Yaskawa INFORM job: MALBEN3.JBI

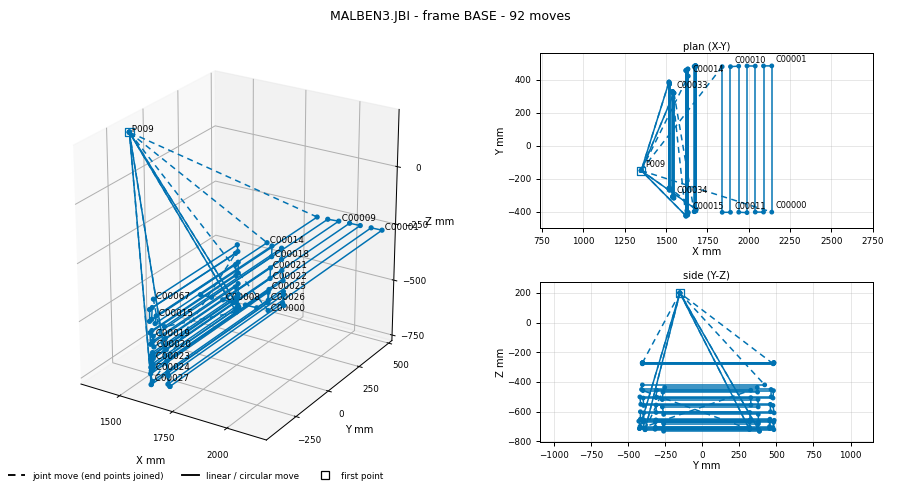
[picture p0: tool path of MALBEN3.JBI in frame BASE, 92 of 92 moves have a stored position in this frame; points joined in program order, loops and branches not executed]
/JOB
//NAME MALBEN3
//POS
///NPOS 86,0,86,1,0,1
///TOOL 0
///POSTYPE BASE
///RECTAN
///RCONF 1,0,0,0,0,0,0,0,0,0,0,0,0,0,0,0,0,0,0,0,0,0,0,0
C00000=2140.098,-401.360,-268.977,175.0000,5.0000,5.0000
C00001=2140.098,483.583,-268.977,175.0000,5.0000,5.0000
C00002=2090.098,483.455,-270.030,175.0000,5.0000,5.0000
C00003=2090.098,-401.273,-270.030,175.0000,5.0000,5.0000
C00004=2040.098,-401.141,-271.239,175.0000,5.0000,5.0000
C00005=2040.098,482.568,-271.239,175.0000,5.0000,5.0000
C00006=1990.098,483.262,-272.654,175.0000,5.0000,5.0000
C00007=1990.098,-404.579,-272.654,175.0000,5.0000,5.0000
C00008=1940.098,-401.886,-274.425,175.0000,5.0000,5.0000
C00009=1940.098,482.155,-274.425,175.0000,5.0000,5.0000
C00010=1890.098,478.954,-276.250,175.0000,5.0000,5.0000
C00011=1890.098,-402.510,-276.250,175.0000,5.0000,5.0000
C00012=1839.960,-402.553,-277.742,175.0000,5.0000,5.0000
C00013=1839.960,478.937,-277.742,175.0000,5.0000,5.0000
C00014=1634.901,421.672,-419.637,175.0000,-89.9999,5.0000
C00015=1634.901,-402.743,-419.637,175.0000,-89.9999,5.0000
C00016=1633.143,-408.452,-450.789,175.0000,-89.9999,5.0000
C00017=1633.143,464.348,-450.789,175.0000,-89.9999,5.0000
C00018=1631.374,465.131,-500.789,175.0000,-89.9999,5.0000
C00019=1631.374,-419.852,-500.789,175.0000,-89.9999,5.0000
C00020=1629.352,-413.747,-550.789,175.0000,-89.9999,5.0000
C00021=1629.352,459.427,-550.789,175.0000,-89.9999,5.0000
C00022=1626.911,460.715,-600.789,175.0000,-89.9999,5.0000
C00023=1626.911,-416.191,-600.789,175.0000,-89.9999,5.0000
C00024=1624.499,-416.100,-650.789,175.0000,-89.9999,5.0000
C00025=1624.499,456.978,-650.789,175.0000,-89.9999,5.0000
C00026=1622.503,454.505,-700.789,175.0000,-89.9999,5.0000
C00027=1622.503,-418.968,-700.789,175.0000,-89.9999,5.0000
C00028=1620.879,-427.008,-664.187,180.0000,-60.0000,0.0000
C00029=1620.879,455.687,-664.187,180.0000,-60.0000,0.0000
C00030=1619.373,455.631,-714.187,180.0000,-60.0000,0.0000
C00031=1619.373,-422.309,-714.187,180.0000,-60.0000,0.0000
C00032=1619.373,-422.309,-714.187,180.0000,-60.0000,0.0000
C00033=1538.648,327.998,-455.742,175.0000,-89.9999,5.0000
C00034=1538.648,-307.231,-455.742,175.0000,-89.9999,5.0000
C00035=1539.732,-310.347,-505.742,175.0000,-89.9999,5.0000
C00036=1539.732,327.893,-505.742,175.0000,-89.9999,5.0000
C00037=1540.970,328.259,-555.742,175.0000,-89.9999,5.0000
C00038=1540.970,-310.206,-555.742,175.0000,-89.9999,5.0000
C00039=1542.330,-310.096,-605.742,175.0000,-89.9999,5.0000
C00040=1542.330,320.907,-605.742,175.0000,-89.9999,5.0000
C00041=1543.566,323.502,-655.742,175.0000,-89.9999,5.0000
C00042=1543.566,-311.381,-655.742,175.0000,-89.9999,5.0000
C00043=1545.116,-315.143,-705.742,175.0000,-89.9999,5.0000
C00044=1545.116,319.629,-705.742,175.0000,-89.9999,5.0000
C00045=1546.765,320.274,-669.140,180.0000,-60.0000,0.0000
C00046=1546.765,-315.233,-669.140,180.0000,-60.0000,0.0000
C00047=1548.154,-316.980,-719.140,180.0000,-60.0000,0.0000
C00048=1548.154,319.087,-719.140,180.0000,-60.0000,0.0000
C00049=1548.154,319.087,-719.140,180.0000,-60.0000,0.0000
C00050=1670.216,-398.864,-458.454,175.0000,-89.9999,5.0000
C00051=1670.216,480.762,-458.454,175.0000,-89.9999,5.0000
C00052=1672.445,477.562,-508.454,175.0000,-89.9999,5.0000
C00053=1672.445,-397.223,-508.454,175.0000,-89.9999,5.0000
C00054=1674.551,-394.686,-558.454,175.0000,-89.9999,5.0000
C00055=1674.551,477.382,-558.454,175.0000,-89.9999,5.0000
C00056=1676.296,485.126,-608.454,175.0000,-89.9999,5.0000
C00057=1676.296,-393.486,-608.454,175.0000,-89.9999,5.0000
C00058=1677.899,-392.919,-658.454,175.0000,-89.9999,5.0000
C00059=1677.899,485.748,-658.454,175.0000,-89.9999,5.0000
C00060=1679.509,477.056,-708.454,175.0000,-89.9999,5.0000
C00061=1679.509,-394.482,-708.454,175.0000,-89.9999,5.0000
C00062=1680.701,-393.512,-671.851,180.0000,-60.0000,0.0000
C00063=1680.701,481.956,-671.851,180.0000,-60.0000,0.0000
C00064=1682.129,483.373,-721.851,180.0000,-60.0000,0.0000
C00065=1682.129,-384.577,-721.851,180.0000,-60.0000,0.0000
C00066=1682.129,-384.577,-721.851,180.0000,-60.0000,0.0000
C00067=1520.388,-252.750,-437.009,175.0000,-89.9999,5.0000
C00068=1520.388,371.413,-437.009,175.0000,-89.9999,5.0000
C00069=1521.796,373.507,-468.529,175.0000,-89.9999,5.0000
C00070=1521.796,-264.209,-468.529,175.0000,-89.9999,5.0000
C00071=1521.398,-268.886,-518.529,175.0000,-89.9999,5.0000
C00072=1521.398,376.643,-518.529,175.0000,-89.9999,5.0000
C00073=1521.017,377.744,-568.529,175.0000,-89.9999,5.0000
C00074=1521.017,-268.182,-568.529,175.0000,-89.9999,5.0000
C00075=1519.841,-259.271,-618.529,175.0000,-89.9999,5.0000
C00076=1519.841,378.499,-618.529,175.0000,-89.9999,5.0000
C00077=1519.405,379.693,-668.529,175.0000,-89.9999,5.0000
C00078=1519.405,-263.625,-668.529,175.0000,-89.9999,5.0000
C00079=1519.161,-262.870,-718.529,175.0000,-89.9999,5.0000
C00080=1519.161,378.578,-718.529,175.0000,-89.9999,5.0000
C00081=1518.693,379.125,-681.927,180.0000,-60.0000,0.0000
C00082=1518.693,-258.984,-681.927,180.0000,-60.0000,0.0000
C00083=1518.160,-259.608,-731.927,180.0000,-60.0000,0.0000
C00084=1518.160,386.235,-731.927,180.0000,-60.0000,0.0000
C00085=1518.160,386.235,-731.927,180.0000,-60.0000,0.0000
///POSTYPE PULSE
///PULSE
EC00000=0
EC00001=0
EC00002=0
EC00003=0
EC00004=0
EC00005=0
EC00006=0
EC00007=0
EC00008=0
EC00009=0
EC00010=0
EC00011=0
EC00012=0
EC00013=0
EC00014=0
EC00015=0
EC00016=0
EC00017=0
EC00018=0
EC00019=0
EC00020=0
EC00021=0
EC00022=0
EC00023=0
EC00024=0
EC00025=0
EC00026=0
EC00027=0
EC00028=0
EC00029=0
EC00030=0
EC00031=0
EC00032=92160
EC00033=92160
EC00034=92160
EC00035=92160
EC00036=92160
EC00037=92160
EC00038=92160
EC00039=92160
EC00040=92160
EC00041=92160
EC00042=92160
EC00043=92160
EC00044=92160
EC00045=92160
EC00046=92160
EC00047=92160
EC00048=92160
EC00049=184320
EC00050=184320
EC00051=184320
EC00052=184320
EC00053=184320
EC00054=184320
EC00055=184320
EC00056=184320
EC00057=184320
EC00058=184320
EC00059=184320
EC00060=184320
EC00061=184320
EC00062=184320
EC00063=184320
EC00064=184320
EC00065=184320
EC00066=276480
EC00067=276480
EC00068=276480
EC00069=276480
EC00070=276480
EC00071=276480
EC00072=276480
EC00073=276480
EC00074=276480
EC00075=276480
EC00076=276480
EC00077=276480
EC00078=276480
EC00079=276480
EC00080=276480
EC00081=276480
EC00082=276480
EC00083=276480
EC00084=276480
EC00085=368640
///POSTYPE BASE
///RECTAN
P00009=1350.000,-150.000,200.000,-180.0000,-45.0000,0.0000
///POSTYPE PULSE
///PULSE
EX00000=0
//INST
///DATE 2023/03/14 16:30
///ATTR SC,RW,RJ
////FRAME BASE
///GROUP1 RB1,ST1
NOP
MOVJ P009 EX000 VJ=15.00
MOVJ C00000 EC00000 VJ=15.00
CALL JOB:SPYON
MOVL C00001 EC00001 V=150.0
MOVL C00002 EC00002 V=150.0
MOVL C00003 EC00003 V=150.0
MOVL C00004 EC00004 V=150.0
MOVL C00005 EC00005 V=150.0
MOVL C00006 EC00006 V=150.0
MOVL C00007 EC00007 V=150.0
MOVL C00008 EC00008 V=150.0
MOVL C00009 EC00009 V=150.0
MOVL C00010 EC00010 V=150.0
MOVL C00011 EC00011 V=150.0
MOVL C00012 EC00012 V=150.0
MOVL C00013 EC00013 V=150.0
CALL JOB:SPYOF
MOVJ P009 VJ=15.00
MOVJ C00014 EC00014 VJ=15.00
CALL JOB:SPYON
MOVL C00015 EC00015 V=150.0
MOVL C00016 EC00016 V=150.0
MOVL C00017 EC00017 V=150.0
MOVL C00018 EC00018 V=150.0
MOVL C00019 EC00019 V=150.0
MOVL C00020 EC00020 V=150.0
MOVL C00021 EC00021 V=150.0
MOVL C00022 EC00022 V=150.0
MOVL C00023 EC00023 V=150.0
MOVL C00024 EC00024 V=150.0
MOVL C00025 EC00025 V=150.0
MOVL C00026 EC00026 V=150.0
MOVL C00027 EC00027 V=150.0
MOVL C00028 EC00028 V=150.0
MOVL C00029 EC00029 V=150.0
MOVL C00030 EC00030 V=150.0
MOVL C00031 EC00031 V=150.0
CALL JOB:SPYOF
MOVJ P009 VJ=15.00
MOVL C00032 EC00032 V=150.0
MOVJ C00033 EC00033 VJ=15.00
CALL JOB:SPYON
MOVL C00034 EC00034 V=150.0
MOVL C00035 EC00035 V=150.0
MOVL C00036 EC00036 V=150.0
MOVL C00037 EC00037 V=150.0
MOVL C00038 EC00038 V=150.0
MOVL C00039 EC00039 V=150.0
MOVL C00040 EC00040 V=150.0
MOVL C00041 EC00041 V=150.0
MOVL C00042 EC00042 V=150.0
MOVL C00043 EC00043 V=150.0
MOVL C00044 EC00044 V=150.0
MOVL C00045 EC00045 V=150.0
MOVL C00046 EC00046 V=150.0
MOVL C00047 EC00047 V=150.0
MOVL C00048 EC00048 V=150.0
CALL JOB:SPYOF
MOVJ P009 VJ=15.00
MOVL C00049 EC00049 V=150.0
MOVJ C00050 EC00050 VJ=15.00
CALL JOB:SPYON
MOVL C00051 EC00051 V=150.0
MOVL C00052 EC00052 V=150.0
MOVL C00053 EC00053 V=150.0
MOVL C00054 EC00054 V=150.0
MOVL C00055 EC00055 V=150.0
MOVL C00056 EC00056 V=150.0
MOVL C00057 EC00057 V=150.0
MOVL C00058 EC00058 V=150.0
MOVL C00059 EC00059 V=150.0
MOVL C00060 EC00060 V=150.0
MOVL C00061 EC00061 V=150.0
MOVL C00062 EC00062 V=150.0
MOVL C00063 EC00063 V=150.0
MOVL C00064 EC00064 V=150.0
MOVL C00065 EC00065 V=150.0
CALL JOB:SPYOF
MOVJ P009 VJ=15.00
MOVL C00066 EC00066 V=150.0
MOVJ C00067 EC00067 VJ=15.00
CALL JOB:SPYON
MOVL C00068 EC00068 V=150.0
MOVL C00069 EC00069 V=150.0
MOVL C00070 EC00070 V=150.0
MOVL C00071 EC00071 V=150.0
MOVL C00072 EC00072 V=150.0
MOVL C00073 EC00073 V=150.0
MOVL C00074 EC00074 V=150.0
MOVL C00075 EC00075 V=150.0
MOVL C00076 EC00076 V=150.0
MOVL C00077 EC00077 V=150.0
MOVL C00078 EC00078 V=150.0
MOVL C00079 EC00079 V=150.0
MOVL C00080 EC00080 V=150.0
MOVL C00081 EC00081 V=150.0
MOVL C00082 EC00082 V=150.0
MOVL C00083 EC00083 V=150.0
MOVL C00084 EC00084 V=150.0
CALL JOB:SPYOF
MOVJ P009 VJ=15.00
MOVL C00085 EC00085 V=150.0
END
